TYPE T_Char : STRING[1];
END_TYPE

(* stored: Version 1.1.0.1
   DUT T_Char: Id {30cb7c55-5bb9-4f02-bde1-7f86c5c91f4b} *)
